// TIA Portal V17 export
// export: Created 2024-10-17T14:16:15.3458547Z, ExportSetting WithDefaults, DisplayName Totally Integrated Automation Portal, DisplayVersion V17 Update 4, DisplayName TIA Portal Openness, DisplayVersion V17 Update 4, DisplayName TIA Portal Version Control Interface, DisplayVersion V17, DisplayName SINAMICS Startdrive Advanced, DisplayVersion V17 Update2, DisplayName SINAMICS Startdrive G130, G150, S120, S150, SINAMICS MV, S210, DisplayVersion V17 Update2, DisplayName SINAMICS Startdrive G110M, G120, G120C, G120D, G120P, G115D, DisplayVersion V17 Update2, DisplayName STEP 7 Professional, DisplayVersion V17 Update 4, DisplayName STEP 7 Safety, DisplayVersion V17, DisplayName WinCC Advanced / Unified PC, DisplayVersion V17 Update 4
DATA_BLOCK "InstLPMLV2022_Stacklight"   // DB30113
{ DB_Accessible_From_OPC_UA := 'FALSE' }
AUTHOR : APC_ERLF
FAMILY : OMAC
VERSION : 1.0
// stored: AutoNumber true, DBAccessibleFromOPCUA false, DBAccessibleFromWebserver false, InstanceOfName LPMLV2022_Stacklight, InstanceOfType FB
"LPMLV2022_Stacklight"
   // VAR_INPUT
   //    StateCurrent : DInt;
   //    starvedUpstream : Bool;
   //    blockedDownstream : Bool;
   //    materialLow : Bool;
   //    materialExhausted : Bool;
   // END_VAR
   // VAR_OUTPUT
   //    Stacklight { ExternalWritable := 'False'} : DWord;
   //    redSolid { ExternalWritable := 'False'} : Bool;
   //    redFlashing { ExternalWritable := 'False'} : Bool;
   //    amberSolid { ExternalWritable := 'False'} : Bool;
   //    amberFlashing { ExternalWritable := 'False'} : Bool;
   //    blueSolid { ExternalWritable := 'False'} : Bool;
   //    blueFlashing { ExternalWritable := 'False'} : Bool;
   //    greenSolid { ExternalWritable := 'False'} : Bool;
   //    greenFlashing { ExternalWritable := 'False'} : Bool;
   //    hornFlashing { ExternalWritable := 'False'} : Bool;
   // END_VAR
BEGIN
END_DATA_BLOCK
